// TIA Portal project "bottle_conveyor_sytem" (V17)
// This a program to simulate industrial bottling using a HMI and TIA

(* hardware
DEVICE "HMI_1"  KTP700 Basic PN
   slot 0: "HMI_1"  KTP700 Basic PN  6AV2 123-2GB03-0AX0  15.1.0.0
   slot 1: "HMI_RT_1"  KTP700 Basic PN  6AV2 123-2GB03-0AX0  15.1.0.0
   slot 5: "HMI_1.IE_CP_1"  PROFINET Interface  15.0.1.0
      slot 1: "PROFINET Interface_1"  PROFINET Interface
         slot 1: "Port_1"  Port
DEVICE "S7-1200 station_1"  S7-1200 Station
   slot 0: "Rack_0"  S7-1200 Rack  Rack  V1.0
   slot 1: "PLC_1"  CPU 1214C DC/DC/DC  6ES7 214-1AG40-0XB0  V4.0
*)

// ===== PLC "PLC_1"  CPU 1214C DC/DC/DC =====

VAR_GLOBAL   // PLC tag table "Default tag table"
   "start_button" AT %M0.0 : Bool;
   "stop_button" AT %M0.1 : Bool;
   "conveyor" AT %Q0.0 : Bool;
END_VAR

ORGANIZATION_BLOCK "Main"   // OB1, LAD, ProgramCycle
TITLE = "Main Program Sweep (Cycle)"
{ S7_Optimized_Access := 'TRUE' }
VERSION : 0.1
   VAR_INPUT
      Initial_Call : Bool;   // Initial call of this OB
      Remanence : Bool;   // =True, if remanent data are available
   END_VAR
BEGIN

REGION Network 1
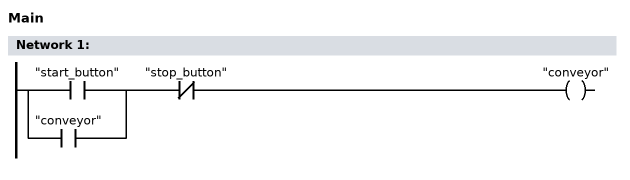
   RUNG wire#powerrail
      Contact( "start_button" )
      wire#w1
      I_Contact( "stop_button" )
      Coil( "conveyor" )
   END_RUNG
   RUNG wire#powerrail
      Contact( "conveyor" )
   END_RUNG wire#w1
   // the same network as SCL:
   "conveyor" := ("start_button" OR "conveyor") AND NOT "stop_button";
END_REGION
END_ORGANIZATION_BLOCK

(* ===== HMI "HMI_RT_1" =====
system functions are stored by id; their names below are inferred from use
connection "HMI_Connection_1": ETHERNET, SMART_S7_1200_OMS

HMI tags "Default tag table"
   "start_button" : Bool = PLC start_button AT %M0.0, 1 s
   "stop_button" : Bool = PLC stop_button AT %M0.1, 1 s
   "move" : Int, internal
   "conveyor" : Bool = PLC conveyor AT %Q0.0, 1 s

screen "Screen_1" 800x480
   on GenerateScreen: function_f9c01323("move", 1, 100, 0, 1)
   Button "Button_1" at 1,13 size 255x45; TextOff 'Automatic'
   Button "Button_2" at 0,70 size 258x51; TextOff 'Manual'
   Button "Button_3" at 3,418 size 191x45; TextOff 'Start'
      on Press: SetBit("start_button")
      on Release: ResetBit("start_button")
   Button "Button_4" at 221,419 size 188x52; TextOff 'Stop'
      on Press: SetBit("stop_button")
      on Release: ResetBit("stop_button")
   GraphicView "Graphic view_3" at 64,277 size 560x40; Picture "Graphic_3"
   GraphicView "Graphic view_1" at 71,136 size 68x169; Picture "Graphic_1"
      HorizontalMovement <- "move"
      Visibility <- "conveyor"
   Group "Group" at 672,322 size 120x150
   Group "Group_1" at 764,443 size 24x24
   Group "Group_2" at 734,443 size 24x24
   Group "Group_3" at 705,443 size 24x24
   Group "Group_4" at 675,443 size 24x24
   Group "Group_5" at 675,413 size 24x24
   Group "Group_6" at 705,414 size 24x24
   Group "Group_7" at 734,414 size 24x24
   Group "Group_8" at 764,413 size 24x24
   Group "Group_9" at 764,384 size 24x24
   Group "Group_10" at 734,384 size 24x24
   Group "Group_11" at 704,384 size 24x24
   Group "Group_12" at 675,384 size 24x24
   Group "Group_13" at 764,356 size 24x24
   Group "Group_14" at 734,356 size 24x24
   Group "Group_15" at 704,356 size 24x24
   Group "Group_16" at 675,356 size 24x24
   Group "Group_17" at 764,328 size 24x24
   Group "Group_18" at 734,327 size 24x24
   Group "Group_19" at 705,328 size 24x24
   Group "Group_20" at 675,327 size 24x24
   Button "Button_5" at 549,4 size 232x54; TextOff 'New box'
*)